PROGRAM main
VAR
	Start_Btn AT %IX0.0 : bool;
	Stop_Btn AT %IX0.1 : bool;
	System_Active AT %QX0.0 : bool;
END_VAR

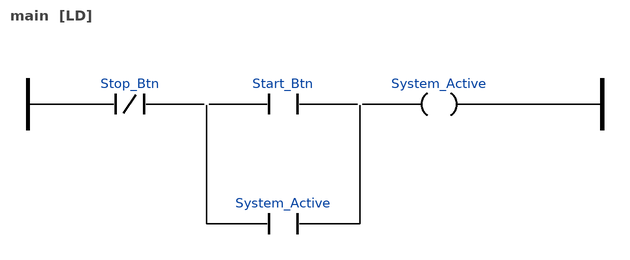
(* LD diagram, written out as Structured Text *)
System_Active := NOT Stop_Btn AND (Start_Btn OR System_Active);
END_PROGRAM
